// Represents the current serialization state and is passed along
// as the serialization proceeds.
// All the public methods are intended to be invoked only by the generated code,
// users should never invoke them directly.
{attribute 'no_explicit_call' := 'do not call this POU directly'} 
FUNCTION_BLOCK PUBLIC FINAL FB_WriteContext
VAR
    stCtx   : ST_WriteContext;
END_VAR

VAR
END_VAR

METHOD FromBuffer : HRESULT
VAR_IN_OUT CONSTANT
    aBuffer : ARRAY [*] OF BYTE;
END_VAR

Reset();
Initialize(F_SpanFromArray(aBuffer));
END_METHOD

METHOD INTERNAL Initialize
VAR_INPUT CONSTANT
    stBuffer    : ST_Span;    
END_VAR
stCtx.stBuffer := stBuffer;

stCtx.stState.nBufferSize        := stBuffer.nSize;
stCtx.stState.nBufferPos         := 0;

stCtx.pCurrentContext			:= THIS;
END_METHOD

// Initialize a ST_WriterContext using existing ST_WriterInternalState,
METHOD INTERNAL InitializeFromState
VAR_IN_OUT CONSTANT
    stBuffer : ST_Span;
    stState : ST_WriterInternalState;        
END_VAR
THIS^.stCtx.stState  := stState;
THIS^.stCtx.stBuffer := stBuffer;

stCtx.pCurrentContext := THIS;
END_METHOD

PROPERTY nSpaceLeft : UDINT
GET
nSpaceLeft := stCtx.stState.nBufferSize - stCtx.stState.nBufferPos;
END_GET
END_PROPERTY

PROPERTY refCtx : REFERENCE TO ST_WriteContext
GET
refCtx REF= THIS^.stCtx ;
END_GET
END_PROPERTY

METHOD PRIVATE Reset
VAR_INPUT
END_VAR

stCtx.stState.bError := FALSE;
stCtx.stState.eWriterErrorCode := S_OK;
stCtx.stState.nBufferPos := 0;
stCtx.stState.nBufferSize := 0;
END_METHOD

METHOD WriteBool : HRESULT
VAR_INPUT
    bValue : BOOL;
END_VAR

WriteBool := F_WriteRawByte(THIS^.stCtx, TO_BYTE(bValue));
END_METHOD

METHOD WriteBytes : HRESULT
VAR_IN_OUT CONSTANT
    aBytes  : ARRAY [*] OF BYTE;
END_VAR
VAR_INPUT
    nCount : UDINT;
END_VAR

WriteBytes := F_WriteBytes(THIS^.stCtx, aBytes, nCount);
END_METHOD

METHOD WriteDouble : HRESULT
VAR_INPUT
    fValue : LREAL;
END_VAR
WriteDouble := F_WriteDouble(THIS^.stCtx, fValue);
END_METHOD

METHOD WriteEnum : HRESULT
VAR_INPUT
    anyEnum : ANY;
END_VAR
VAR
	nTmp : DINT;
END_VAR
IF anyEnum.pValue = NULL OR anyEnum.TypeClass <> __SYSTEM.TYPE_CLASS.TYPE_ENUM THEN
	WriteEnum := E_HRESULTAdsErr.INVALIDDATA;
	RETURN;
END_IF

MEMCPY(destAddr:= ADR(nTmp), srcAddr:= anyEnum.pValue, MIN(TO_UDINT(anyEnum.diSize), SIZEOF(nTmp)));
WriteEnum := F_WriteEnum(THIS^.stCtx, nTmp);
END_METHOD

METHOD WriteFixed32 : HRESULT
VAR_INPUT
    nValue : UDINT;
END_VAR

WriteFixed32 := F_WriteFixed32(THIS^.stCtx, nValue);
END_METHOD

METHOD WriteFixed64 : HRESULT
VAR_INPUT
    nValue : ULINT;
END_VAR

WriteFixed64 := F_WriteFixed64(THIS^.stCtx, nValue);
END_METHOD

METHOD WriteFloat : HRESULT
VAR_INPUT
    fValue : REAL;
END_VAR
WriteFloat := F_WriteFloat(THIS^.stCtx, fValue);
END_METHOD

METHOD WriteInt32 : HRESULT
VAR_INPUT
    anyDint : ANY;
END_VAR
VAR
    nTmp   : DINT;
	retVal : UDINT;
END_VAR

retVal := memcpy(destAddr:= ADR(nTmp), srcAddr:= anyDint.pValue, n:= MIN(TO_UDINT(anyDint.diSize), SIZEOF(nTmp)));
IF retVal = 0 THEN
	WriteInt32:= E_HRESULTAdsErr.INVALIDDATA;
	RETURN;
END_IF

WriteInt32 := F_WriteInt32(THIS^.stCtx, nTmp);
END_METHOD

METHOD WriteInt64 : HRESULT
VAR_INPUT
    anyLint : ANY;
END_VAR
VAR
    nTmp   : LINT;
	retVal : UDINT;
END_VAR

retVal := memcpy(destAddr:= ADR(nTmp), srcAddr:= anyLint.pValue, n:= MIN(TO_UDINT(anyLint.diSize), SIZEOF(nTmp)));
IF retVal = 0 THEN
	WriteInt64:= E_HRESULTAdsErr.INVALIDDATA;
	RETURN;
END_IF

WriteInt64 := F_WriteInt64(THIS^.stCtx, nTmp);
END_METHOD

METHOD WriteLength : HRESULT
VAR_INPUT
    nLength : UDINT;
END_VAR

WriteLength := F_WriteLength(THIS^.stCtx, nLength);
END_METHOD

METHOD WriteMessage : HRESULT
VAR_INPUT
    ipMessage : I_Message;
END_VAR

WriteMessage := F_WriteMessage(stCtx:= THIS^.stCtx, ipMessage);
END_METHOD

METHOD WriteRawTag : HRESULT
VAR_INPUT
	nTag    : UDINT;
END_VAR
WriteRawTag := F_WriteRawTag(THIS^.stCtx, nTag);
END_METHOD

METHOD WriteSFixed32 : HRESULT
VAR_INPUT
    nValue : DINT;
END_VAR

WriteSFixed32 := F_WriteSFixed32(THIS^.stCtx, nValue);
END_METHOD

METHOD WriteSFixed64 : HRESULT
VAR_INPUT
    nValue : LINT;
END_VAR

WriteSFixed64 := F_WriteSFixed64(THIS^.stCtx, nValue);
END_METHOD

METHOD WriteSint32 : HRESULT
VAR_INPUT
    anyDint : ANY;
END_VAR
VAR
    nTmp   : DINT;
	retVal : UDINT;
END_VAR

retVal := memcpy(destAddr:= ADR(nTmp), srcAddr:= anyDint.pValue, n:= MIN(TO_UDINT(anyDint.diSize), SIZEOF(nTmp)));
IF retVal = 0 THEN
	WriteSint32:= E_HRESULTAdsErr.INVALIDDATA;
	RETURN;
END_IF

WriteSint32 := F_WriteSInt32(THIS^.stCtx, nTmp);
END_METHOD

METHOD WriteSint64 : HRESULT
VAR_INPUT
    anyLint : ANY;
END_VAR
VAR
    nTmp   : LINT;
	retVal : UDINT;
END_VAR

retVal := memcpy(destAddr:= ADR(nTmp), srcAddr:= anyLint.pValue, n:= MIN(TO_UDINT(anyLint.diSize), SIZEOF(nTmp)));
IF retVal = 0 THEN
	WriteSint64:= E_HRESULTAdsErr.INVALIDDATA;
	RETURN;
END_IF

WriteSint64 := F_WriteSInt64(THIS^.stCtx, nTmp);
END_METHOD

METHOD WriteString : HRESULT
VAR_IN_OUT CONSTANT
    sStringToWrite          : T_ProtobufMaxString;
END_VAR

WriteString := F_WriteString(THIS^.stCtx, sStringToWrite);
END_METHOD

METHOD WriteTag : HRESULT
VAR_INPUT
    nFieldNumber    : UDINT;
    eWireType       : E_WireType;
END_VAR

WriteTag := F_WriteTag(THIS^.stCtx, nFieldNumber, eWireType);
END_METHOD

METHOD WriteUint32 : HRESULT
VAR_INPUT
    anyUdint : ANY;
END_VAR
VAR
    nTmp   : UDINT;
	retVal : UDINT;
END_VAR


retVal := memcpy(destAddr:= ADR(nTmp), srcAddr:= anyUdint.pValue, n:= MIN(TO_UDINT(anyUdint.diSize), SIZEOF(nTmp)));
IF retVal = 0 THEN
	WriteUint32:= E_HRESULTAdsErr.INVALIDDATA;
	RETURN;
END_IF

WriteUint32 := F_WriteUInt32(THIS^.stCtx, nTmp);
END_METHOD

METHOD WriteUint64 : HRESULT
VAR_INPUT
    anyUlint : ANY;
END_VAR
VAR
    nTmp   : ULINT;
	retVal : UDINT;
END_VAR

retVal := memcpy(destAddr:= ADR(nTmp), srcAddr:= anyUlint.pValue, n:= MIN(TO_UDINT(anyUlint.diSize), SIZEOF(nTmp)));
IF retVal = 0 THEN
	WriteUint64:= E_HRESULTAdsErr.INVALIDDATA;
	RETURN;
END_IF

WriteUint64 := F_WriteUInt64(THIS^.stCtx, nTmp);
END_METHOD

END_FUNCTION_BLOCK

(* stored: Version 1.1.0.1
   POU FB_WriteContext: Id {18246595-6bbb-43ef-aa75-24f9e22ace2b}, SpecialFunc None
   Method FromBuffer: Id {1e98a2df-1c25-4299-8859-723e4bc10e7e}
   Method Initialize: Id {29caada7-8387-4211-be03-001b7a8625e2}
   Method InitializeFromState: Id {e95638a0-ab7e-4b84-941e-d84723767bdb}
   Property nSpaceLeft: Id {81be7da9-2e5d-48e4-88e3-0f185cdb7127}
   Get Get: Id {060dd1c8-d1ad-424e-8a91-006db807548b}
   Property refCtx: Id {e5294272-b90e-41bf-a1d1-aff26b19e5fd}
   Get Get: Id {b80681af-b361-4c87-8d39-73970893001f}
   Method Reset: Id {7023c71a-5838-4abb-a6b6-612b36e632a1}
   Method WriteBool: Id {959509b8-b6ba-41cc-a129-8f0ea33bc2ff}
   Method WriteBytes: Id {02b8f0af-661f-4944-85ff-f76fd4cec3ea}
   Method WriteDouble: Id {3b86ec3f-2cad-45c5-9a6f-d56de79d1415}
   Method WriteEnum: Id {4fb9d4ab-4be6-42ee-a3bb-3f86dbf2061c}
   Method WriteFixed32: Id {75c23fcd-723d-4cbc-9e77-8e2301b57ac1}
   Method WriteFixed64: Id {ac5b07e1-2d27-4aea-84db-e2a22552a9fb}
   Method WriteFloat: Id {ec5060f6-e490-4798-a185-1d013ad3518c}
   Method WriteInt32: Id {cb424f8c-2286-402b-adff-21634a582503}
   Method WriteInt64: Id {470d349f-a883-451f-86ff-5add09c6bbc1}
   Method WriteLength: Id {aefabf76-233a-48e5-bd46-c3bd214198fb}
   Method WriteMessage: Id {9347cb0b-4bb2-4141-9235-78ef0ba3ee66}
   Method WriteRawTag: Id {a86dd6ed-09e8-4909-8291-9a826323973b}
   Method WriteSFixed32: Id {c5db7557-6b1a-4521-ab52-97e9e0d0670f}
   Method WriteSFixed64: Id {1d1909aa-43d1-452a-93e7-9bb5567d60cd}
   Method WriteSint32: Id {9b3c1ae8-a598-4a54-9dcf-fc39ef583879}
   Method WriteSint64: Id {b35dcafc-ac19-4012-a560-388617eee3d1}
   Method WriteString: Id {e0704046-198b-43d6-993d-44c5595830da}
   Method WriteTag: Id {7d0d5de0-234e-4fd9-b783-7b62ad087c0a}
   Method WriteUint32: Id {5d55f154-a20b-441b-9140-093b322d95f5}
   Method WriteUint64: Id {340b2f1b-3da7-48bf-82ca-67d4a8315258} *)
